{attribute 'qualified_only'}
VAR_GLOBAL
	(* Digital IO to Byte *)
	aDigitalInputIO AT %I* 	: ARRAY[1..9]OF BYTE; //KL1408 9EA
	aDigitalOutputIO AT %Q* : ARRAY[1..5]OF BYTE; //KL2408 4EA
	
	(* Analog Input to INT*)
	aAnalogInputIO AT %I* 	: ARRAY[1..40] OF INT;
	aAnalogOutputIO AT %Q* 	: ARRAY[1..40] OF INT;
	aAnalogInputIO2 AT %I*	: ARRAY[1..2]OF UINT;
	
	(*Solenoid Valve*)
	aOutputSolValve AT %Q* 	: DWORD; //Solenoid Valve
	
	(* Read and Write of Device Control Value*)
	aMaxValueController		: ARRAY[1..GVL_CONSTANT.NumAnalogController] OF REAL ; //Device Max Value from UI
	aController 			: ARRAY[1..GVL_CONSTANT.NumAnalogController] OF FB_ControlRampGenerator; //MFC, EPC 0 ~ 5V
	aController_PV 			: ARRAY[1..GVL_CONSTANT.NumAnalogController] OF REAL; //Present Value from Device
	aController_CV 			: ARRAY[1..GVL_CONSTANT.NumAnalogController] OF REAL; //Current Value from RampingController
	
	(* Present Value Meter Display*)
	aMonitoring_PV 			: ARRAY[1..17] OF REAL; //Gauge Monitoring Value to UI
	aInputState				: ARRAY[1..6] OF WORD; // Digital Input from Device (Switch)
	aOutputCmd				: ARRAY[1..3] OF WORD; // Digital Command from UI
	aInterlock				: ARRAY[1..5] OF DWORD; // Interlock
	aInterlockSet			: ARRAY[1..16] OF REAL; // UI Interlokc Setting Value
	aInterlockEnable		: ARRAY[1..6] OF DWORD; // UI Interlock Enable Setting
	
	//jhkang
//	aInterlock_Alarm: ARRAY[1..E_AlarmList.E_AlarmList_END]OF BOOL;// Interlock
//	aInterlock_Warning: ARRAY[1..E_WarningList.E_WarningList_END]OF BOOL;// Interlock
//	aInterlock_jh:ARRAY[1..E_Interlock.E_Interlock_END]OF BOOL;
//	aInterlockSet_jh: ARRAY[1..E_AlarmSetValue.E_AS_END] OF REAL; // UI Interlokc Setting Value
//	aInterlockEnable_jh:ARRAY[1..6]OF BOOL;
	
	nCaseSignalTower		: INT;
	nDorOperationError		: INT;
	bDorState				: BOOL;
	bDorOnEnable			: BOOL;
// 	bE3508_HeaterOn			: BOOL;
	wE3508_CV				: WORD;
	wE3508_PV				: WORD;
	wIqPlus_CV				: WORD;
	wIqPlus_CDG1_PV			: WORD;
	wIqPlus_CDG2_PV			: WORD;
	nRotation_Converted_PV	: INT;
	rRotation_ControlValue	: REAL;
	nIQPLUS_SetType 		: INT;
	nIQPLUS_Mode			: INT;
	aLineHeater_rTemperaturePV : ARRAY[1..8]OF REAL;
	nE3508_nInputManAutoBytes : USINT;
	isCoverClosed 			: BOOL;
	isPumpRunning 			: BOOL;
END_VAR

(* stored: Version 1.1.0.1, ProductVersion 3.1.4026.11
   GVL GVL_IO: Id {a5f3292d-798a-4b6c-af88-b59309d83086} *)
